(* IEC 61131-3 sources: Industry-PLC-LLM/data/PLCBEAD_repo/PLCBEAD_PLCEmbed-main/PLC-BEAD/Source/GEB/Network_TN_SC_XY_ERROR, 1 file *)

(* ---- TN_SC_XY_ERROR.ST ---- *)
FUNCTION TN_SC_XY_ERROR:BOOL

	VAR_INPUT
		X :	INT;
		Y :	INT;
	END_VAR

	TN_SC_XY_ERROR := Y < 0 OR X < 0 OR Y > 23 OR X > 79;

END_FUNCTION

PROGRAM program0
	VAR
		X :	INT;
		Y :	INT;
		CEIL5_OUT : BOOL;
	END_VAR

  	CEIL5_OUT := TN_SC_XY_ERROR(X, Y);
END_PROGRAM
